FUNCTION_BLOCK DSCYL_MDLL (* Model for a Double-Stroke Cylinder, Externally Clocked *)
  (* Standard: 61499-1 *)
  (* Version 0.1, 2004-10-20, JHC, Rockwell Automation, Added UNLD, REND_ID, LOAD_ID, LOAD_SUB, LOADER. *)
  (* Version 0.0, 2004-09-25, JHC, Rockwell Automation, Extended from DSCYL_MDL1. *)
  (* Compiler header: package fb.rt.mach; import fb.rt.net.*; import fb.rt.mva.*; *)
  (* Compiler classdef: public class DSCYL_MDLL extends FBMVCD *)
  (* Compiler Java Sun JDK 1.4.2 *)
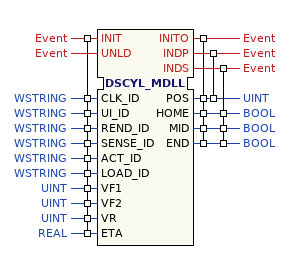
  EVENT_INPUT
    INIT WITH ACT_ID, CLK_ID, UI_ID, SENSE_ID, VF1, VF2, VR, ETA, LOAD_ID, REND_ID; (* Initialize *)
    UNLD;
  END_EVENT
  EVENT_OUTPUT
    INITO WITH POS, HOME, MID, END;
    INDP WITH POS; (* Position Change Indication *)
    INDS WITH HOME, MID, END; (* Sensor Change Indication *)
  END_EVENT
  VAR_INPUT
    CLK_ID : WSTRING := "SIM_CLK"; (* Simulation clock channel ID *)
    UI_ID : WSTRING; (* User input channel ID from View *)
    REND_ID : WSTRING; (* Local Channel ID for Rendering Data *)
    SENSE_ID : WSTRING; (* Sensor data channel ID to Controller *)
    ACT_ID : WSTRING; (* Actuator data channel ID from Controller *)
    LOAD_ID : WSTRING; (* Loader data channel ID for WKPC+STYLE *)
    VF1 : UINT; (* Cyl#1 ADVANCE speed in %FS per CLK event *)
    VF2 : UINT; (* Cyl#2 ADVANCE speed in %FS per CLK event *)
    VR : UINT; (* RETRACT speed in %FS per CLK event *)
    ETA : REAL := 0.5; (* Length ratio:Cyl#1/(Cyl#1+Cyl#2) *)
  END_VAR
  VAR_OUTPUT
    POS : UINT; (* End effector position *)
    HOME : BOOL; (* Both cylinders HOME *)
    MID : BOOL; (* CYL1 at END,CYL2 HOME *)
    END : BOOL; (* Both cylinders at END *)
  END_VAR
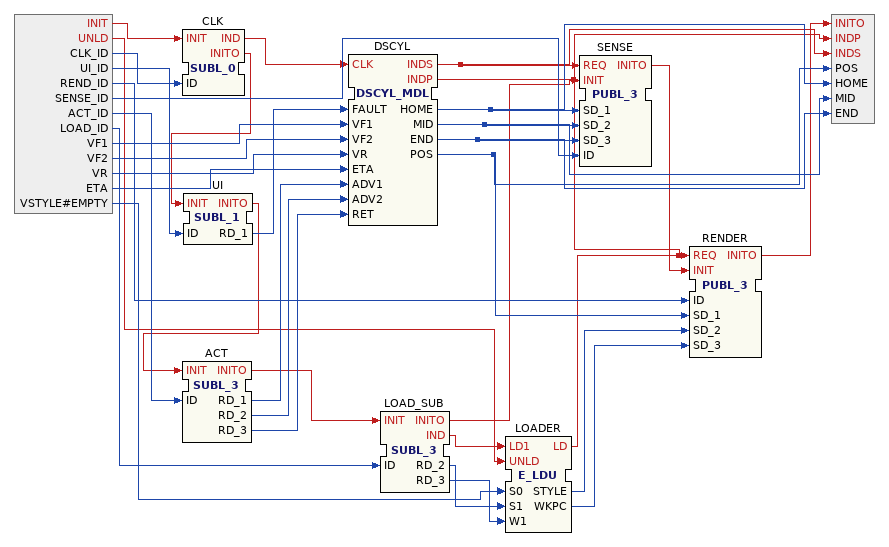
  FBS
    DSCYL : DSCYL_MDL;
    CLK : SUBL_0;
    UI : SUBL_1;
    SENSE : PUBL_3;
    ACT : SUBL_3;
    LOADER : E_LDU;
    LOAD_SUB : SUBL_3;
    RENDER : PUBL_3;
  END_FBS
  EVENT_CONNECTIONS
    INIT TO CLK.INIT;
    CLK.IND TO DSCYL.CLK;
    CLK.INITO TO UI.INIT;
    DSCYL.INDS TO SENSE.REQ;
    UI.INITO TO ACT.INIT;
    DSCYL.INDP TO INDP;
    DSCYL.INDS TO INDS;
    ACT.INITO TO LOAD_SUB.INIT;
    LOAD_SUB.INITO TO SENSE.INIT;
    LOAD_SUB.IND TO LOADER.LD1;
    LOADER.LD TO RENDER.REQ;
    SENSE.INITO TO RENDER.INIT;
    RENDER.INITO TO INITO;
    UNLD TO LOADER.UNLD;
    DSCYL.INDP TO RENDER.REQ;
  END_CONNECTIONS
  DATA_CONNECTIONS
    UI.RD_1 TO DSCYL.FAULT;
    VF1 TO DSCYL.VF1;
    VF2 TO DSCYL.VF2;
    VR TO DSCYL.VR;
    ETA TO DSCYL.ETA;
    DSCYL.HOME TO SENSE.SD_1;
    DSCYL.MID TO SENSE.SD_2;
    DSCYL.END TO SENSE.SD_3;
    DSCYL.HOME TO HOME;
    DSCYL.MID TO MID;
    DSCYL.END TO END;
    ACT.RD_1 TO DSCYL.ADV1;
    ACT.RD_2 TO DSCYL.ADV2;
    ACT.RD_3 TO DSCYL.RET;
    SENSE_ID TO SENSE.ID;
    CLK_ID TO CLK.ID;
    UI_ID TO UI.ID;
    ACT_ID TO ACT.ID;
    LOAD_ID TO LOAD_SUB.ID;
    REND_ID TO RENDER.ID;
    DSCYL.POS TO RENDER.SD_1;
    LOADER.STYLE TO RENDER.SD_2;
    LOADER.WKPC TO RENDER.SD_3;
    VSTYLE#EMPTY TO LOADER.S0;
    DSCYL.POS TO POS;
    LOAD_SUB.RD_2 TO LOADER.S1;
    LOAD_SUB.RD_3 TO LOADER.W1;
  END_CONNECTIONS
END_FUNCTION_BLOCK
